FUNCTION_BLOCK GetArrayResponseFromJSON (* Transfor a HTTP response to an array *)
  (* Standard: 61499-2; Description: Copyright (c) 2018 fortiss GmbH This program and the accompanying materials are made available under the terms of the Eclipse Public License 2.0 which is available at https://www.eclipse.org/legal/epl-2.0/ SPDX-License-Identifier: EPL-2.0 *)
  (* Version 1.0, 2018-09-21, Jose Cabral, fortiss GmbH *)
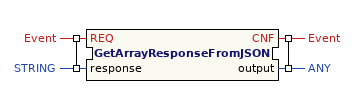
  EVENT_INPUT
    REQ WITH response; (* Request response from HTTP *)
  END_EVENT
  EVENT_OUTPUT
    CNF WITH output; (* Response requested *)
  END_EVENT
  VAR_INPUT
    response : STRING; (* Reponse from HTTP *)
  END_VAR
  VAR_OUTPUT
    output : ANY; (* Ouptut result *)
  END_VAR
  (* Service APPLICATION/RESOURCE: Transfor a HTTP response to an array *)
END_FUNCTION_BLOCK
